// TIA Portal V20 export
TYPE "LWONIK_typeFromSafetyDoorStatus"
// stored: Access Published
   STRUCT
      FdoorSwitchStatus { ExternalWritable := 'False'} : Struct
         unwinderRearDoorOpen : Bool;
         autoSpliceDoorOpen : Bool;
         unwinderMainDoorOpen : Bool;
         unwinderTopDoorOpen : Bool;
         unwinderBtmDoorOpen : Bool;
         StackTableDoorOpen : Bool;
         winderDoorOpen : Bool;
      END_STRUCT;
      FdoorCoilStatus { ExternalWritable := 'False'} : Struct
         unwinderRearDoorUnlock : Bool;
         autoSpliceDoorUnlock : Bool;
         unwinderMainDoorUnlock : Bool;
         unwinderTopDoorUnlock : Bool;
         unwinderBtmDoorUnlock : Bool;
         StackTableDoorUnlock : Bool;
         winderDoorUnlock : Bool;
      END_STRUCT;
   END_STRUCT;
END_TYPE
